// LS Electric XG5000 project: 동남115
// PLC NewPLC
// module base 0 slot 0: 입출력 모듈:XBC-DN/DP14E (DC 24V 입력 8점, 트랜지스터 출력 6점)

PROGRAM NewProgram (task: 스캔 프로그램)

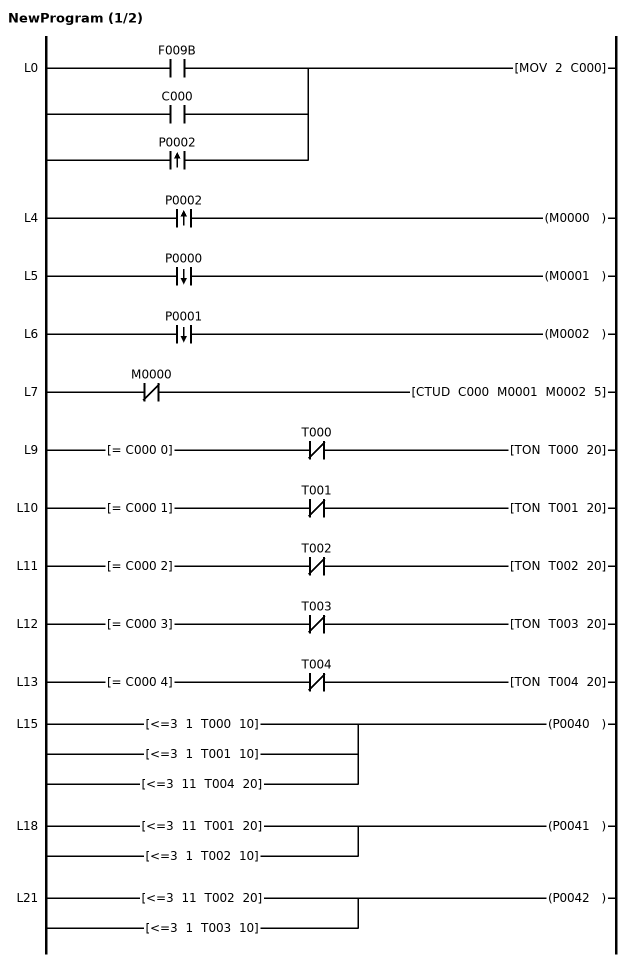
; L0
LOAD      F009B
OR        C000
ORP       P0002
MOV       2 C000
; L4
LOADP     P0002
OUT       M0000
; L5
LOADN     P0000
OUT       M0001
; L6
LOADN     P0001
OUT       M0002
; L7
LOAD NOT  M0000
CTUD      C000 M0001 M0002 5
; L9
LOAD=     C000 0
AND NOT   T000
TON       T000 20
; L10
LOAD=     C000 1
AND NOT   T001
TON       T001 20
; L11
LOAD=     C000 2
AND NOT   T002
TON       T002 20
; L12
LOAD=     C000 3
AND NOT   T003
TON       T003 20
; L13
LOAD=     C000 4
AND NOT   T004
TON       T004 20
; L15
LOAD<=3   1 T000 10
OR<=3     1 T001 10
OR<=3     11 T004 20
OUT       P0040
; L18
LOAD<=3   11 T001 20
OR<=3     1 T002 10
OUT       P0041
; L21
LOAD<=3   11 T002 20
OR<=3     1 T003 10
OUT       P0042

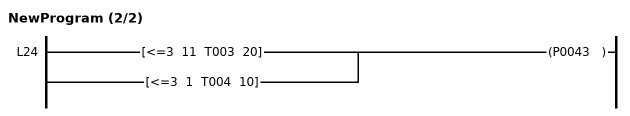
; L24
LOAD<=3   11 T003 20
OR<=3     1 T004 10
OUT       P0043